// TIA Portal V17 export
// export: Created 2022-04-06T07:28:38.4932328Z, ExportSetting WithDefaults, DisplayName Totally Integrated Automation Portal, DisplayVersion V17, DisplayName TIA Portal Openness, DisplayVersion V17, DisplayName TIA Portal Version Control Interface, DisplayVersion V17, DisplayName TIA Portal Test Suite Advanced, DisplayVersion V17, DisplayName SINAMICS Startdrive Advanced, DisplayVersion V17, DisplayName SINAMICS Startdrive G130, G150, S120, S150, SINAMICS MV, S210, DisplayVersion V17, DisplayName SINAMICS Startdrive G110M, G120, G120C, G120D, G120P, G115D, DisplayVersion V17, DisplayName STEP 7 Professional, DisplayVersion V17, DisplayName STEP 7 Safety, DisplayVersion V17, DisplayName WinCC Advanced / Unified PC, DisplayVersion V17
FUNCTION_BLOCK "SINA_FFB"   // FB5, F_FBD
{ S7_Optimized_Access := 'TRUE' }
VERSION : 0.1
// stored: AutoNumber true, IsIECCheckEnabled true, UDAEnableTagReadback false
   VAR_INPUT
      tel30Status : "LDrvSafe_typeSinaSTlg30Status";
      acknowledge : Bool;
      releaseEstop : Bool := true;
      releaseGate : Bool := true;
      enableMode : Bool := true;
   END_VAR
   VAR_OUTPUT
      tel30Control : "LDrvSafe_typeSinaSTlg30Control";
   END_VAR
   VAR
      statSlsTof : TOF;
      statTrue : Bool;
   END_VAR
BEGIN

REGION Network 1
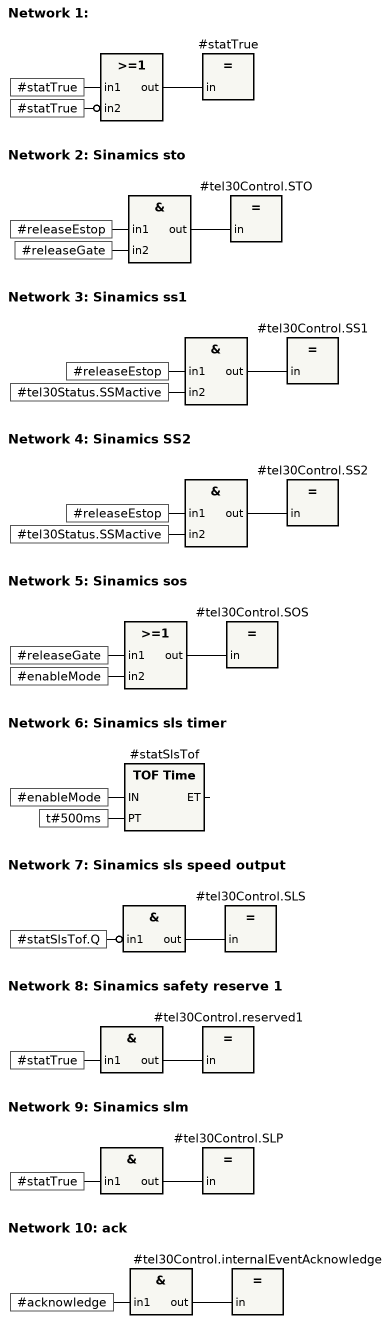
   #statTrue := #statTrue OR NOT #statTrue;
END_REGION

REGION Network 2: Sinamics sto
   #tel30Control.STO := #releaseEstop AND #releaseGate;
END_REGION

REGION Network 3: Sinamics ss1
   #tel30Control.SS1 := #releaseEstop AND #tel30Status.SSMactive;
END_REGION

REGION Network 4: Sinamics SS2
   #tel30Control.SS2 := #releaseEstop AND #tel30Status.SSMactive;
END_REGION

REGION Network 5: Sinamics sos
   #tel30Control.SOS := #releaseGate OR #enableMode;
END_REGION

REGION Network 6: Sinamics sls timer
   #statSlsTof.TOF(IN := #enableMode, PT := t#500ms);
END_REGION

REGION Network 7: Sinamics sls speed output
   #tel30Control.SLS := NOT #statSlsTof.Q;
END_REGION

REGION Network 8: Sinamics safety reserve 1
   #tel30Control.reserved1 := #statTrue;
END_REGION

REGION Network 9: Sinamics slm
   #tel30Control.SLP := #statTrue;
END_REGION

REGION Network 10: ack
   #tel30Control.internalEventAcknowledge := #acknowledge;
END_REGION

REGION Network 11: Sinamics safety reserve 2
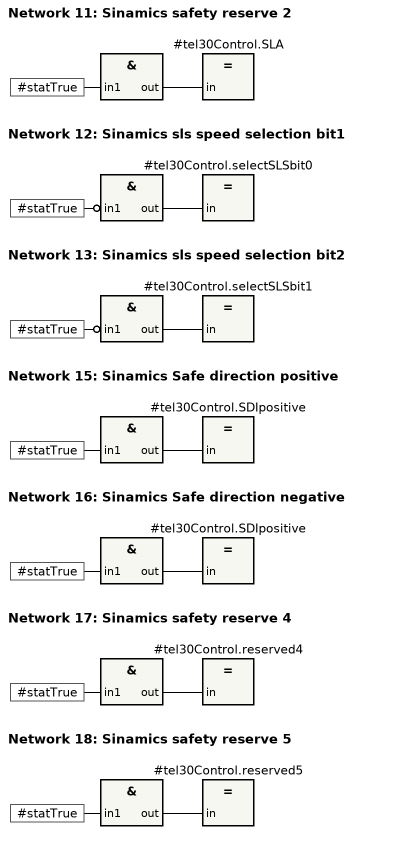
   #tel30Control.SLA := #statTrue;
END_REGION

REGION Network 12: Sinamics sls speed selection bit1
   #tel30Control.selectSLSbit0 := NOT #statTrue;
END_REGION

REGION Network 13: Sinamics sls speed selection bit2
   #tel30Control.selectSLSbit1 := NOT #statTrue;
END_REGION

REGION Network 14: Sinamics safety reserve 3
END_REGION

REGION Network 15: Sinamics Safe direction positive
   #tel30Control.SDIpositive := #statTrue;
END_REGION

REGION Network 16: Sinamics Safe direction negative
   #tel30Control.SDIpositive := #statTrue;
END_REGION

REGION Network 17: Sinamics safety reserve 4
   #tel30Control.reserved4 := #statTrue;
END_REGION

REGION Network 18: Sinamics safety reserve 5
   #tel30Control.reserved5 := #statTrue;
END_REGION
END_FUNCTION_BLOCK
